Yaskawa INFORM job: TEST_ABOVE.JBI

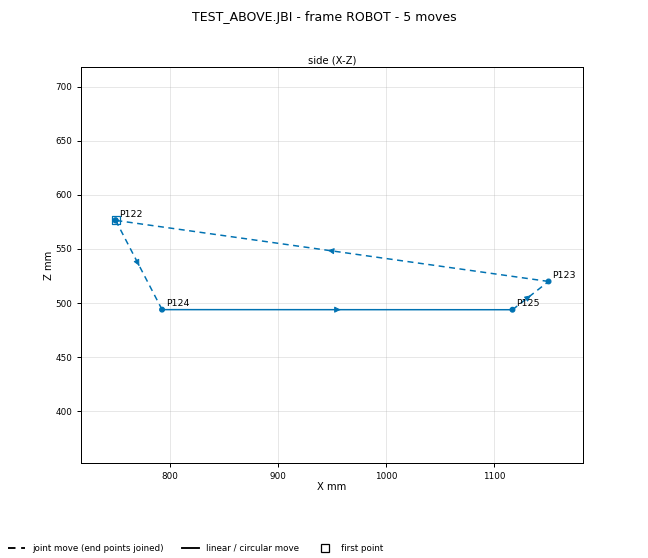
[picture p0: tool path of TEST_ABOVE.JBI in frame ROBOT, 5 of 5 moves have a stored position in this frame; points joined in program order, loops and branches not executed]
/JOB
//NAME TEST_ABOVE
///FOLDERNAME FOLDER001
//POS
///NPOS 2,0,0,4,0,0
///USER 15
///TOOL 1
///POSTYPE USER
///RECTAN
///RCONF 1,0,0,0,0,0,0,0,0,0,0,0,0,0,0,0,0,0,0,0,0,0,0,0
C00000=4.666,-1.318,179.409,180.0000,-10.0000,0.0000
C00001=4.513,-65.064,179.402,180.0000,-10.0000,0.0000
///POSTYPE ROBOT
P00122=750.004,162.000,576.437,180.0000,-9.9968,0.0000
P00123=1150.002,160.000,520.003,180.0000,-25.0002,0.0000
P00124=792.896,161.791,493.972,179.9986,-9.9993,0.0008
P00125=1116.664,160.780,493.887,-179.9993,-9.9981,-0.0025
//INST
///DATE 2025/09/30 14:27
///ATTR SC,RW,RJ
////FRAME USER 15
///GROUP1 RB1
///LVARS 20,20,20,0,0,0,0,0
NOP
SFTOF
MACRO1 MJ#(2) ARGF2.4 ARGF1.0 ARGF0.0
MACRO1 MJ#(1) ARGF0.0 ARGF0.0 ARGF0.0 ARGF0.0 ARGF0.0 ARGF0.0
REFP 1 C00000
REFP 2 C00001
MOVJ P122 VJ=15.00 PL=3
MOVJ P124 VJ=15.00 PL=0
WVON AMP=D080 FREQ=D081 ANGL=D082
WVADJ STD=4.000 ST=4.000 END=4.000 LEN=400.000 ADJMD=0
MOVL P125 V=25.0 PL=0
WVOF
MOVJ P123 VJ=15.00 PL=3
MOVJ P122 VJ=15.00 PL=3
SFTOF
END
